KUKA KRL program: style1app1opt2A.src, style1app1opt2A.dat

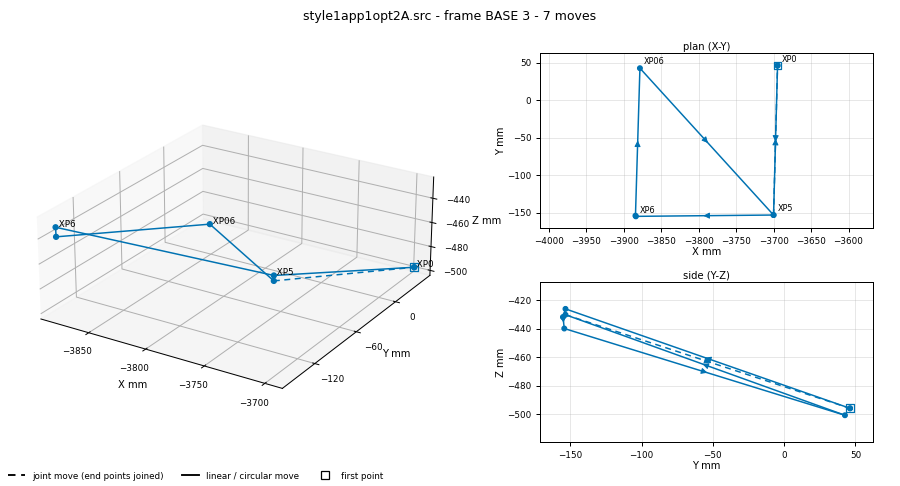
[picture p0: tool path of style1app1opt2A.src in frame BASE 3, 7 of 7 moves have a stored position in this frame; points joined in program order, loops and branches not executed]
--- style1app1opt2A.src ---
&ACCESS RVO1
&REL 246
&COMMENT 03-10-R1 PNW1 NUT 2 ST1
&PARAM EDITMASK = *
&PARAM TEMPLATE = C:\KRC\TP\Nutweld\Template\NutWeld_Vorgabe
&PARAM DISKPATH = KRC:\R1\Program\StyleApps\Options
DEF style1app1opt2A( )
   ;FOLD INI
      ;FOLD BASISTECH INI
         GLOBAL INTERRUPT DECL 3 WHEN $STOPMESS==TRUE DO IR_STOPM ( )
         INTERRUPT ON 3
         BAS (#INITMOV,0 )
      ;ENDFOLD (BASISTECH INI)
      ;FOLD NutWeld
      ;ENDFOLD (NutWeld)
      ;FOLD USER INI
         ;Make your modifications here

      ;ENDFOLD (USER INI)
   ;ENDFOLD (INI)
;********************************
; Gestamp Standards
; Line - BMW G65 (cell 03)
; Robot 03-10-R1 (BMW-03-10-R1-PNW1)
; Application - WELD NUT 2 (PN2) AT THE CENTERLINE PEDESTAL - PART FROM PICKUP 1 (A)
;********************************
; CALLED BY Style1Opt1. APPROACH THE PEDESTAL (BASE 3 "NUT WELDER"), WAIT FOR THE NUT PRELOAD
; (NEXT_NUT_READY), MOVE THE PART TO THE WELD POSITION P16, WELD WITH CENTERLINE_WELD (NOT IN DRY
; CYCLE), LEAVE THE PEDESTAL.
;WARNING: BEFORE THE ROBOT MOVES IN, GUN OPEN, SUBMIT AND WATER ARE CHECKED (GUN_OPEN_CHECK) -
;  NOT CLAMP OPEN OR QFP RETURNED (F01)
;NOTE: THE PEDESTAL MOVES MIX BASE MODE AND EXTERNAL-TCP MODE (extTCP); THE WELD POSITION
;  P16 IS TAUGHT IN BASE MODE (F22)
;APPROACH THE PEDESTAL - P0, P5
;FOLD PTP P0 CONT Vel=100 % PDAT0 Tool[1]:TOOL 1 Base[3]:NUT WELDER extTCP;%{PE}%R 8.3.43,%MKUKATPBASIS,%CMOVE,%VPTP,%P 1:PTP, 2:P0, 3:C_DIS, 5:100, 7:PDAT0
$BWDSTART=FALSE
PDAT_ACT=PPDAT0
FDAT_ACT=FP0
BAS(#PTP_PARAMS,100)
PTP XP0 C_DIS
;ENDFOLD
;FOLD LIN P5 Vel=2 m/s CPDAT11 Tool[1]:TOOL 1 Base[3]:NUT WELDER;%{PE}%R 8.3.43,%MKUKATPBASIS,%CMOVE,%VLIN,%P 1:LIN, 2:P5, 3:, 5:2, 7:CPDAT11
$BWDSTART=FALSE
LDAT_ACT=LCPDAT11
FDAT_ACT=FP5
BAS(#CP_PARAMS,2)
LIN XP5
;ENDFOLD
;GUN MONITORING - INTERRUPTS 20-22 CALL GUN_OPEN_LOST (BRAKE F, QUIT MESSAGE) WHEN THE GUN LEAVES THE
;OPEN RANGE (CL_GunStrokePositionLPT 137000..142000) OR THE SUBMIT STOPS WHILE THE ROBOT MOVES INTO
;OR OUT OF THE PEDESTAL. EDGE TRIGGERED: GUN_OPEN_CHECK CONFIRMS THE GUN OPEN AFTER EVERY ON (F01)
;WARNING: THE RANGE IS WRITTEN HERE AS LITERALS; KEEP IT EQUAL TO nGunOpenMin/nGunOpenMax IN
;  GUN_OPEN_CHECK.dat (F01)
INTERRUPT DECL 20 WHEN CL_GunStrokePositionLPT<137000 DO GUN_OPEN_LOST()
INTERRUPT DECL 21 WHEN CL_GunStrokePositionLPT>142000 DO GUN_OPEN_LOST()
INTERRUPT DECL 22 WHEN $PRO_STATE0<>#P_ACTIVE DO GUN_OPEN_LOST()
;CYCLE-TIME MEASUREMENT (NO EFFECT ON THE SEQUENCE): ROBOT STOPPED AT THE WAIT POINT (WAIT SEC 0),
;$TIMER[20] FROM HERE FOR NUT 2 (CL_CYCLE_TIME, F52)
WAIT SEC 0
CL_CYCLE_START(2)
;WAIT NUT PRELOADED - NEXT_NUT_READY (SET WHEN THE PRELOAD ENDS, QFP SEEN RETURNED; NO NUT SENSOR,
;  F13)
;NOTE: NO TIMEOUT, NO MESSAGE (F15). IN DRY CYCLE NOTHING SETS IT: THE CYCLE HANGS HERE (F04)
WAIT FOR NEXT_NUT_READY==TRUE
;CYCLE-TIME MARK - STEP 1 NUT READY (CL_CYCLE_TIME, F52)
CL_CYCLE_TIME(1)
;FEED NUT 3 INTO THE SHUTTLE NOW, WHILE THE ROBOT MOVES IN AND WELDS: THE SHUTTLE IS RETURNED
;AND EMPTY, NUT 2 IS ON THE PIN. PRELOAD ONLY FEEDS; IT LOADS NUT 3 ONTO THE PIN WHEN
;Request_next_nut IS CALLED AT P05 ON THE WAY OUT. ONLY WITH NO PRELOAD RUNNING AND OUTSIDE DRY CYCLE
;(SIGNAL $IN[4] di004UseDryCycle OFF) - ELSE Request_next_nut FEEDS AND LOADS AS BEFORE (F52)
IF NUT_READY AND NOT NUTCYCLE_ACTIVE AND NOT di004UseDryCycle THEN
   NUT_FEED_START=TRUE
ENDIF
;GUN MONITORING ON FIRST (THE INTERRUPTS FIRE ONLY ON A CHANGE), THEN THE INTERLOCK: GUN OPEN,
;SUBMIT RUNNING, WATER OK (GUN_OPEN_CHECK); THE MONITORING STAYS ON WHILE THE ROBOT MOVES IN (F01)
INTERRUPT ON 20
INTERRUPT ON 21
INTERRUPT ON 22
GUN_OPEN_CHECK()
;MOVE IN - P6 (2 M/S), THEN THE WELD POSITION P16 OUTSIDE DRY CYCLE
;FOLD LIN P6 Vel=2 m/s CPDAT0 Tool[1]:TOOL 1 Base[3]:NUT WELDER;%{PE}%R 8.3.43,%MKUKATPBASIS,%CMOVE,%VLIN,%P 1:LIN, 2:P6, 3:, 5:2, 7:CPDAT0
$BWDSTART=FALSE
LDAT_ACT=LCPDAT0
FDAT_ACT=FP6
BAS(#CP_PARAMS,2)
LIN XP6
;ENDFOLD

;OUTSIDE DRY CYCLE ONLY (SIGNAL $IN[4] di004UseDryCycle OFF): WELD POSITION P16 AND CENTERLINE_WELD()
;NOTE: $IN[4] IS RE-READ AT EVERY STEP; SWITCHED ON MID-CYCLE, THIS NUT IS NOT WELDED AND
;  THE PART CAN STILL REACH THE GOOD DROP (F05)
IF NOT di004UseDryCycle THEN
;FOLD LIN P16 Vel=2 m/s CPDAT15 Tool[1]:TOOL 1 Base[3]:NUT WELDER;%{PE}%R 8.3.43,%MKUKATPBASIS,%CMOVE,%VLIN,%P 1:LIN, 2:P16, 3:, 5:2, 7:CPDAT15
$BWDSTART=FALSE
LDAT_ACT=LCPDAT15
FDAT_ACT=FP16
BAS(#CP_PARAMS,2)
LIN XP16
;ENDFOLD
;ROBOT AT THE WELD POSITION (WAIT SEC 0 STOPS THE ADVANCE RUN): GUN MONITORING OFF, THE GUN
;CLOSES ON PURPOSE IN CENTERLINE_WELD
WAIT SEC 0
INTERRUPT OFF 20
INTERRUPT OFF 21
INTERRUPT OFF 22
;NUT WELD AT THE PEDESTAL (CENTERLINE_WELD: CLAMP, GUN, INTENSIFY, BOSCH WELD, GUN OPEN)
CENTERLINE_WELD()
;GUN MONITORING ON WHILE LEAVING, THEN THE GUN OPEN IS CONFIRMED AGAIN (GUN_OPEN_CHECK): A GUN THAT
;LEFT THE OPEN RANGE AFTER THE CHECK INSIDE CENTERLINE_WELD WOULD NOT TRIGGER THE INTERRUPTS (F01)
INTERRUPT ON 20
INTERRUPT ON 21
INTERRUPT ON 22
GUN_OPEN_CHECK()
ENDIF
;LEAVE THE PEDESTAL - P06, P05, P0 (THE DRY CYCLE CONTINUES HERE)
;FOLD LIN P06 CONT Vel=2 m/s CPDAT6 Tool[1]:TOOL 1 Base[3]:NUT WELDER extTCP;%{PE}%R 8.3.43,%MKUKATPBASIS,%CMOVE,%VLIN,%P 1:LIN, 2:P06, 3:C_DIS C_DIS, 5:2, 7:CPDAT6
$BWDSTART=FALSE
LDAT_ACT=LCPDAT6
FDAT_ACT=FP06
BAS(#CP_PARAMS,2)
LIN XP06 C_DIS C_DIS
;ENDFOLD
;ROBOT OUT OF THE PEDESTAL (WAIT SEC 0 STOPS THE ADVANCE RUN, NO APPROXIMATION HERE): GUN
;MONITORING OFF
WAIT SEC 0
INTERRUPT OFF 20
INTERRUPT OFF 21
INTERRUPT OFF 22
;FOLD LIN P05 Vel=2 m/s CPDAT14 Tool[1]:TOOL 1 Base[3]:NUT WELDER;%{PE}%R 8.3.43,%MKUKATPBASIS,%CMOVE,%VLIN,%P 1:LIN, 2:P05, 3:, 5:2, 7:CPDAT14
$BWDSTART=FALSE
LDAT_ACT=LCPDAT14
FDAT_ACT=FP05
BAS(#CP_PARAMS,2)
LIN XP05
;ENDFOLD
;NEXT NUT - TRIGGER ON THE MOTION TO P0 (DISTANCE = 0: FIRES WHEN THE MOTION STARTS, AT P05 - EXACT
;STOP - PRIO -1). P05 IS 4 MM FROM P5, WHERE THE ROBOT ALREADY WAITS WHILE THE QFP LOADS NUT 2
;(WAS DISTANCE = 1, AT P0). Request_next_nut() CLEARS NEXT_NUT_READY AND SETS NUT_START: PRELOAD
;LOADS NUT 3 (FED DURING THE WELD) ONTO THE PIN, OR FEEDS AND LOADS IT IF NOTHING WAS FED (F52)
;NOTE: THE TRIGGER STANDS BEFORE THE INLINE FORM, SO A TOUCH UP OF P0 CANNOT DELETE IT; IT ACTS ON
;  THE NEXT MOTION. A BLOCK SELECTION ONTO THE MOTION FOLD SKIPS IT (SELECT THE TRIGGER LINE),
;  AND SO DOES A PROGRAM RESET: NUT 3 THEN WAITS FOR EVER FOR NEXT_NUT_READY (F14, F38)
TRIGGER WHEN DISTANCE = 0 DELAY = 0 DO Request_next_nut() PRIO= -1
;FOLD PTP P0 Vel=100 % PDAT26 Tool[1]:TOOL 1 Base[3]:NUT WELDER extTCP;%{PE}%R 8.3.43,%MKUKATPBASIS,%CMOVE,%VPTP,%P 1:PTP, 2:P0, 3:, 5:100, 7:PDAT26
$BWDSTART=FALSE
PDAT_ACT=PPDAT26
FDAT_ACT=FP0
BAS(#PTP_PARAMS,100)
PTP XP0
;ENDFOLD


END

--- style1app1opt2A.dat ---
&ACCESS RVO1
&REL 246
&COMMENT GE4_002_GUN1
&PARAM EDITMASK = *
&PARAM TEMPLATE = C:\KRC\TP\Nutweld\Template\NutWeld_Vorgabe
&PARAM DISKPATH = KRC:\R1\Program\StyleApps\Options
DEFDAT  style1app1opt2A
;FOLD EXTERNAL DECLARATIONS;%{PE}%MKUKATPBASIS,%CEXT,%VCOMMON,%P
;FOLD BASISTECH EXT;%{PE}%MKUKATPBASIS,%CEXT,%VEXT,%P
EXT  BAS (BAS_COMMAND  :IN,REAL  :IN )
;ENDFOLD (BASISTECH EXT)
;FOLD NutWeld
;ENDFOLD (NutWeld)
;FOLD USER EXT;%{E}%MKUKATPUSER,%CEXT,%VEXT,%P
;Make here your modifications
;ENDFOLD (USER EXT)
;ENDFOLD (EXTERNAL DECLARATIONS)
DECL NutWeld_SUGG_T LAST_NutWeld={POINT1[] "PNW2_SPOT3              ",POINT2[] "PNW0                    ",CP_PARAMS[] "CPDATNutWeld0           ",PTP_PARAMS[] "PDATNutWeld0            ",CONT[] "C_PTP                   ",CP_VEL[] "2                       ",PTP_VEL[] "100                     ",SYNC_PARAMS[] "SYNCDAT                 ",SPL_NAME[] "S0                      ",NutWeld_PARAMS[] "NutData2_3              ",GunNr 2,SpotNr 3,Offset 45}
DECL BASIS_SUGG_T LAST_BASIS={POINT1[] "P0                      ",POINT2[] "P0                      ",CP_PARAMS[] "CPDAT0                  ",PTP_PARAMS[] "PDAT0                   ",CONT[] "                        ",CP_VEL[] "2                       ",PTP_VEL[] " 100                    ",SYNC_PARAMS[] "SYNCDAT                 ",SPL_NAME[] "S0                      ",A_PARAMS[] "ADAT0                   "}
DECL LDAT Lpnw1={VEL 2.00000,ACC 100.000,APO_DIST 100.000,APO_FAC 50.0000,AXIS_VEL 100.000,AXIS_ACC 100.000,ORI_TYP #VAR,CIRC_TYP #BASE,JERK_FAC 50.0000,GEAR_JERK 50.0000,EXAX_IGN 0}
DECL E6POS XPnw1={X -681.099854,Y -933.961731,Z 7.00223589,A -84.9330902,B -1.72864902,C -2.54664612,S 2,T 11,E1 0.0,E2 0.0,E3 0.0,E4 0.0,E5 0.0,E6 0.0}
DECL FDAT FPnw1={TOOL_NO 1,BASE_NO 3,IPO_FRAME #TCP,POINT2[] " ",TQ_STATE FALSE}

DECL PDAT PPDAT0={VEL 100.000,ACC 100.000,APO_DIST 100.000,APO_MODE #CDIS,GEAR_JERK 50.0000,EXAX_IGN 0}
DECL E6POS XP0={X -3694.69214,Y 46.1868858,Z -495.861603,A -178.336945,B 1.01745069,C 179.989838,S 2,T 34,E1 0.0,E2 0.0,E3 0.0,E4 0.0,E5 0.0,E6 0.0}
DECL FDAT FP0={TOOL_NO 1,BASE_NO 3,IPO_FRAME #TCP,POINT2[] " ",TQ_STATE FALSE}
DECL E6POS XP5={X -3700.01831,Y -153.317429,Z -426.154480,A -178.336502,B -1.01672721,C 179.960312,S 2,T 34,E1 0.0,E2 0.0,E3 0.0,E4 0.0,E5 0.0,E6 0.0}
DECL FDAT FP5={TOOL_NO 1,BASE_NO 3,IPO_FRAME #BASE,POINT2[] " ",TQ_STATE FALSE}
DECL LDAT LCPDAT0={VEL 2.00000,ACC 100.000,APO_DIST 100.000,APO_FAC 50.0000,AXIS_VEL 100.000,AXIS_ACC 100.000,ORI_TYP #VAR,CIRC_TYP #BASE,JERK_FAC 50.0000,GEAR_JERK 50.0000,EXAX_IGN 0}
DECL E6POS XP6={X -3883.74512,Y -155.081940,Z -431.860352,A -178.336502,B -1.01672721,C 179.960312,S 2,T 34,E1 0.0,E2 0.0,E3 0.0,E4 0.0,E5 0.0,E6 0.0}
DECL FDAT FP6={TOOL_NO 1,BASE_NO 3,IPO_FRAME #BASE,POINT2[] " ",TQ_STATE FALSE}
DECL E6POS XP06={X -3878.33521,Y 42.6205063,Z -500.728149,A -178.336945,B 1.01745081,C 179.989838,S 2,T 34,E1 0.0,E2 0.0,E3 0.0,E4 0.0,E5 0.0,E6 0.0}
DECL FDAT FP06={TOOL_NO 1,BASE_NO 3,IPO_FRAME #TCP,POINT2[] " ",TQ_STATE FALSE}
DECL E6POS XP05={X -3700.01831,Y -153.317429,Z -430.255676,A -178.336502,B -1.01672721,C 179.960312,S 2,T 34,E1 0.0,E2 0.0,E3 0.0,E4 0.0,E5 0.0,E6 0.0}
DECL FDAT Fp05={TOOL_NO 1,BASE_NO 3,IPO_FRAME #BASE,POINT2[] " ",TQ_STATE FALSE}
DECL LDAT LCPDAT6={VEL 2.00000,ACC 100.000,APO_DIST 2.00000,APO_FAC 50.0000,AXIS_VEL 100.000,AXIS_ACC 100.000,ORI_TYP #VAR,CIRC_TYP #BASE,JERK_FAC 50.0000,GEAR_JERK 50.0000,EXAX_IGN 0}
DECL PDAT PPDAT26={VEL 100.000,ACC 100.000,APO_DIST 100.000,APO_MODE #CDIS,GEAR_JERK 50.0000,EXAX_IGN 0}
DECL LDAT LCPDAT11={VEL 2.00000,ACC 100.000,APO_DIST 100.000,APO_FAC 50.0000,AXIS_VEL 100.000,AXIS_ACC 100.000,ORI_TYP #VAR,CIRC_TYP #BASE,JERK_FAC 50.0000,GEAR_JERK 50.0000,EXAX_IGN 0}
DECL LDAT LCPDAT14={VEL 2.00000,ACC 100.000,APO_DIST 100.000,APO_FAC 50.0000,AXIS_VEL 100.000,AXIS_ACC 100.000,ORI_TYP #VAR,CIRC_TYP #BASE,JERK_FAC 50.0000,GEAR_JERK 50.0000,EXAX_IGN 0}
DECL E6POS XP16={X -3884.30103,Y -154.162430,Z -439.919525,A -178.336502,B -1.01672733,C 179.960312,S 2,T 34,E1 0.0,E2 0.0,E3 0.0,E4 0.0,E5 0.0,E6 0.0}
DECL FDAT FP16={TOOL_NO 1,BASE_NO 3,IPO_FRAME #BASE,POINT2[] " ",TQ_STATE FALSE}
DECL LDAT LCPDAT15={VEL 2.00000,ACC 100.000,APO_DIST 100.000,APO_FAC 50.0000,AXIS_VEL 100.000,AXIS_ACC 100.000,ORI_TYP #VAR,CIRC_TYP #BASE,JERK_FAC 50.0000,GEAR_JERK 50.0000,EXAX_IGN 0}
ENDDAT
